FUNCTION TryConvert_BOOL_TO_USINT : BOOL
VAR_INPUT
	in : BOOL;
	out : REFERENCE TO USINT;
END_VAR

out := BOOL_TO_USINT(in);
TryConvert_BOOL_TO_USINT := TRUE;

END_FUNCTION

(* stored: Version 1.1.0.1, ProductVersion 3.1.4024.12
   POU TryConvert_BOOL_TO_USINT: Id {8c07e4c1-adf0-4102-8f62-740cb8a22e2d}, SpecialFunc None *)
